# B&R Automation Studio project lektion_8_agdp
Automation Studio 4.8.2.72

## Configuration Config1

### Task classes (Cpu.sw)
```
Cyclic#1:
  assignmen2 <- assignment2.prg
Cyclic#4:
  assignmen1 <- assignment1.prg
Binaries: udbdef, FWRules, TCData, sysconf, Role, User, iomap, ashwd, asfw, arconfig, ashwac
Libraries: runtime, astime, asieccon
```

### Hardware
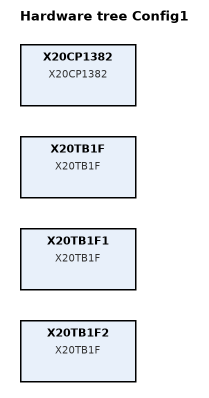
```
X20CP1382 : X20CP1382 v1.10.0.0  [X1 -> X1.SL; X2 -> X2.SL; X3 -> X3.SL]
  Module X1 (Type=X1, Virtual=true, Version=1.10.0.0)
    Connection (Connector=SS1, TargetModule=X20TB1F, TargetConnector=SS)
    Connection (Connector=SL, TargetModule=X20CP1382, TargetConnector=X1)
  Module X2 (Type=X2, Virtual=true, Version=1.10.0.0)
    Connection (Connector=SS1, TargetModule=X20TB1F1, TargetConnector=SS)
    Connection (Connector=SL, TargetModule=X20CP1382, TargetConnector=X2)
  Module X3 (Type=X3, Virtual=true, Version=1.10.0.0)
    Connection (Connector=SS1, TargetModule=X20TB1F2, TargetConnector=SS)
    Connection (Connector=SL, TargetModule=X20CP1382, TargetConnector=X3)
  Connector IF2:
    ActivateDevice = 1
  ConfigurationID = lektion_8_agdp_Config1
  Simulation = 1
X20TB1F : X20TB1F v1.0.0.0
X20TB1F1 : X20TB1F v1.0.0.0
X20TB1F2 : X20TB1F v1.0.0.0
```

## Logical view

### Program Logical/assignment1 (IEC)

#### Variables.var
```iecst
VAR
	RESET : BOOL;
	input : BOOL;
	old_input : BOOL;
	falling_edge : BOOL;
END_VAR
```

#### Main.st
```iecst
PROGRAM _INIT
	(* Insert code here *)
	falling_edge := FALSE;

END_PROGRAM

PROGRAM _CYCLIC
	(* Insert code here *)
//	This does not work correctly
//	IF input = TRUE THEN
//		old_input := FALSE;
//	ELSE
//		old_input := TRUE;
//	END_IF;
//
//	IF input = FALSE AND old_input = TRUE THEN
//		falling_edge := TRUE;
//	ELSE
//		falling_edge := FALSE;
//	END_IF;

//	This works correctly
	IF RESET THEN
		old_input := FALSE;
	ELSE
		falling_edge := old_input AND NOT input;
		old_input := input;
	END_IF;

END_PROGRAM

PROGRAM _EXIT
	(* Insert code here *)

END_PROGRAM
```

### Program Logical/assignment2 (IEC)

#### Variables.var
```iecst
VAR
	doLiftUnload : BOOL;
	doConvLift : BOOL;
	doConvTop : BOOL;
	doConvBot : BOOL;
	doBoxLift : BOOL;
	doLiftBot : BOOL;
	doLiftTop : BOOL;
END_VAR
```

#### Main.st
```iecst
PROGRAM _INIT
	(* Insert code here *)

END_PROGRAM

PROGRAM _CYCLIC
	(* Insert code here *)

	doConvTop    := NOT(doConvBot) AND NOT(doLiftUnload) AND doLiftTop AND NOT(doBoxLift);
	doConvBot    := NOT(doConvTop) AND NOT(doLiftUnload) AND doLiftBot AND NOT(doBoxLift);
	doConvLift   := ((doConvTop OR doConvBot) AND NOT(doBoxLift)) OR (doLiftUnload);
	doLiftTop    := NOT(doLiftBot) AND NOT(doLiftUnload);
	doLiftBot    := NOT(doLiftTop) AND NOT(doLiftUnload);
	doLiftUnload := doBoxLift;

END_PROGRAM

PROGRAM _EXIT
	(* Insert code here *)

END_PROGRAM
```

### Program Logical/assignment2_preben (IEC)

#### Variables.var
```iecst
VAR

	diConvTop : BOOL;

	diConvBottom : BOOL;

	diBoxOnLift : BOOL;

	diLiftTop : BOOL;

	diLiftBottom : BOOL;

	diLiftUnload : BOOL;

	doLiftUnload : BOOL;

	doLiftBottom : BOOL;

	doLiftTop : BOOL;

	doConvBottom : BOOL;

	doConvTop : BOOL;

 END_VAR
```

#### Main.st
```iecst
PROGRAM _INIT
	doConvTop := FALSE;
	doConvBottom := FALSE;
	doLiftTop := FALSE;
	doLiftBottom := FALSE;
	doLiftUnload := FALSE;

 END_PROGRAM

PROGRAM _CYCLIC

 	(* diConvTop : Packagage ready at top lift position *)
 	(* diConvBottom : Packagage ready at bottom lift position *)
 	(* diLiftTop : Lift is at top position *)
 	(* diLiftBottom : Lift is at bottom position *)
 	(* diLiftUnload : Lift is at unload position *)
 	(* diBoxOnLift : Box is on the lift *)

 	// Conveyers kører altid med mindre censor har registreret en pakke
 	// (eller liften er klar til pakke)
	doConvTop := (NOT diConvTop) OR (diLiftTop AND NOT diBoxOnLift AND NOT doLiftBottom);
	doConvBottom := (NOT diConvBottom) OR (diLiftBottom AND NOT diBoxOnLift AND NOT doLiftTop);

	// Hvis der er noget at hente, skal lift køre til top hvis den ikke allerede er på vej et andet sted hen
	// derudover har nederste conveyer første prioritet
	// heri indgår ikke diLiftBottom, da nederste har første prioritet og sensor vil blive
	// aktiveret når den går gennem.
	doLiftTop := (doLiftTop AND NOT diLiftTop) OR (diConvTop AND NOT diLiftTop AND NOT diConvBottom AND NOT doLiftBottom AND NOT doLiftUnload);

	// Samme strategi til nederste, her prioriteres denne dog først
	doLiftBottom := (doLiftBottom AND NOT diLiftBottom) OR (diConvBottom AND NOT diLiftTop AND NOT diLiftBottom AND NOT doLiftTop AND NOT doLiftUnload);

	// Kør til unload position: box på liften
	doLiftUnload := diBoxOnLift;

	// Der mangler logik til at læsse af liften, men dette er ikke en del af opgaven
	// Her "fjerner" vi kassen fra liften

	IF (diLiftUnload) THEN
		diBoxOnLift := FALSE;
	END_IF

 END_PROGRAM

PROGRAM _EXIT
 (* Insert code here *)

 END_PROGRAM
```

Listed in the project but not available here: Logical/Global.typ, Logical/Global.var, Logical/Libraries
